# EPICS autosave request: measCompApp/Db/measCompAnalogInMode_settings.req
$(P)$(R)
